FUNCTION_BLOCK FirstMove
VAR_INPUT
    grab: grab; 
	timer : TP;	
	ccw: moveCCW;
	cw:moveCW;
	down:moveDown;
	iztegni:moveOUT;
	skrci:moveIN;
	up: moveUp;
	relise: relise; 
	itemID: INT := GVL.breadID;
END_VAR
VAR_OUTPUT
	 done: BOOL := FALSE; // Indikator, da je sekvenca zaključena
END_VAR
VAR
	currentState: INT := 0; // Trenutno stanje sekvence
	
	obDol: INT;
	objekt: INT;
	//itemID: INT := 1; //item number
	
	TimerWait: TOF;
	I: INT;
END_VAR

CASE currentState OF
	
	0:
		done := FALSE;
		GVL.downDone := FALSE;
		GVL.grabDone := FALSE;
		currentState := 1;
	
	1:
		down(seconds := T#5S);  // Aktiviraj premik dol
		IF GVL.downDone THEN          // Počakaj, da je premik zaključen
			currentState := 2;     // Premik na naslednje stanje
			GVL.downDone := FALSE;
		END_IF
		
	2:
		grab(seconds := T#2.2S);
		IF GVL.grabDone THEN           // Počakaj, da je prijem zaključen
			currentState := 3;      // Premik na naslednje stanje
			GVL.grabDone := FALSE;
		END_IF
		
	3:
		up(seconds := T#7S);
        IF GVL.upDone THEN           // Počakaj, da je prijem zaključen
            currentState := 4;      // Premik na naslednje stanje
			GVL.upDone := FALSE;
        END_IF

	4:
		//bageta
		IF itemID = 1 THEN
			cw(seconds := T#1.9S);
			IF GVL.CWDone THEN           // Počakaj, da je prijem zaključen
				currentState := 5;      // Premik na naslednje stanje
				GVL.CWDone := FALSE;
			END_IF
		//toast
		ELSIF itemID = 2 THEN
			cw(seconds := T#2.6S);
			IF GVL.CWDone THEN           // Počakaj, da je prijem zaključen
				currentState := 5;      // Premik na naslednje stanje
				GVL.CWDone := FALSE;
			END_IF
		//rženi kruh
		ELSIF itemID = 3 THEN
			cw(seconds := T#3.7S);
			IF GVL.CWDone THEN           // Počakaj, da je prijem zaključen
				currentState := 5;      // Premik na naslednje stanje
				GVL.CWDone := FALSE;
			END_IF
		//bagel
		ELSIF itemID = 4 THEN
			cw(seconds := T#4.2S);
			IF GVL.CWDone THEN           // Počakaj, da je prijem zaključen
				currentState := 5;      // Premik na naslednje stanje
				GVL.CWDone := FALSE;
			END_IF
		END_IF
		
	
	5:
	IF itemID = 1 THEN
		iztegni(seconds := T#4S);
        IF GVL.skrciDone THEN           // Počakaj, da je prijem zaključen
            currentState := 6;      // Premik na naslednje stanje
			GVL.skrciDone := FALSE;
        END_IF
	ELSIF itemID = 2 THEN
		iztegni(seconds := T#2.3S);
        IF GVL.skrciDone THEN           // Počakaj, da je prijem zaključen
            currentState := 6;      // Premik na naslednje stanje
			GVL.skrciDone := FALSE;
        END_IF
	ELSIF itemID = 3 THEN				
		iztegni(seconds := T#2.3S);
        IF GVL.skrciDone THEN           // Počakaj, da je prijem zaključen
            currentState := 6;      // Premik na naslednje stanje
			GVL.skrciDone := FALSE;
        END_IF
	ELSIF itemID = 4 THEN
		iztegni(seconds := T#4.3S);
        IF GVL.skrciDone THEN           // Počakaj, da je prijem zaključen
            currentState := 6;      // Premik na naslednje stanje
			GVL.skrciDone := FALSE;
        END_IF
	END_IF
		
	
	6:
		relise(seconds := T#3S);
        IF GVL.reliseDone THEN           // Počakaj, da je prijem zaključen
            currentState := 7;      // Premik na naslednje stanje
			GVL.reliseDone := FALSE;
        END_IF
	
	7:
		skrci(seconds := T#6S);
        IF GVL.skrciDone THEN           // Počakaj, da je prijem zaključen
            currentState := 8;      // Premik na naslednje stanje
			GVL.skrciDone := FALSE;
        END_IF
	
	8:
		ccw(seconds := T#6S);
        IF GVL.CWDone THEN           // Počakaj, da je prijem zaključen
            //currentState := 9;      // Premik na naslednje stanje
			currentState := 9;
			GVL.CWDone := FALSE;
        END_IF
		
	//9:
	//	GVL.upDone := FALSE;
	//	up(seconds := T#7S);
    //    IF GVL.upDone THEN           // Počakaj, da je prijem zaključen
    //        currentState := 0;      // Premik na naslednje stanje
	//		GVL.upDone := FALSE;
    //    END_IF
	
	 9:
        done := TRUE;               // Označi, da je sekvenca zaključena
        currentState := 0;          // Ponastavi na začetno stanje

	 
END_CASE

END_FUNCTION_BLOCK

(* stored: Version 1.1.0.1, ProductVersion 3.1.4024.15
   POU FirstMove: Id {81f17808-a281-4ee7-8531-e5b869152184}, SpecialFunc None *)
